FUNCTION alg_x: LREAL
{ S7_Optimized_Access := 'true' }
    VAR_INPUT
        state: STATE;
    END_VAR

BEGIN
    alg_x := state.curTime;
END_FUNCTION
